// TIA Portal V20 export
VAR_GLOBAL   // PLC tag table "LAcycCom_Common"
END_VAR
